TYPE ST_LaudaReadCommands_FillLevel :
STRUCT
	BathLevel	: STRING := 'IN_PV_05';
END_STRUCT
END_TYPE

(* stored: Version 1.1.0.1, ProductVersion 3.1.4024.12
   DUT ST_LaudaReadCommands_FillLevel: Id {dbcfdd13-1311-4190-bc7f-ddd8f7543661} *)
